PROGRAM MAIN
VAR
	nIntToRead : INT;
	nIntToWrite : INT;
END_VAR

nIntToRead := nIntToRead + 1;

END_PROGRAM

(* stored: Version 1.1.0.1, ProductVersion 3.1.4024.12
   POU MAIN: Id {c09eab39-212c-4314-9a10-352003bdfd8d}, SpecialFunc None *)
